{attribute 'qualified_only'}
{attribute 'strict'}
{attribute 'to_string'}
TYPE E_ProgressStatus :
(
	Idle,
	Running,
	Paused,
	Completed,
	Error
);
END_TYPE

(* stored: Version 1.1.0.1
   DUT E_ProgressStatus: Id {ae48db73-39c0-4588-9b0d-06202dba6aa2} *)
